TYPE "TMeasuringSts"
VERSION : 0.1
// Block: TMeasuringSts
   STRUCT
      AlarmPresence : Bool;
      InputState : Bool;
      InOperation : Bool;
      MeasuringDone_ID : UInt;
      MeasuringValue1 : LReal;
      MeasuringValue2 : LReal;
   END_STRUCT;

END_TYPE
